// TIA Portal V20 export
DATA_BLOCK "Expedtion"   // DB4
// stored: MemoryReserve 100, Namespace ProductionLine
   VAR
      ExpedtionDirection : Int;
      ExpedtionEnable : Bool;
      CurrentExpedtionDirection : String;
      StraightTableselection : Int;
      CurrentStraightTableselection : String;
      LeftTableselection : Int;
      CurrentLeftTableselection : String;
      StraightTableselectionEnable : Bool;
      LeftTableselectionEnable : Bool;
   END_VAR
BEGIN
END_DATA_BLOCK
